// TIA Portal V17 export
// export: Created 2023-05-31T13:25:21.8623061Z, ExportSetting WithDefaults, DisplayName Totally Integrated Automation Portal, DisplayVersion V17, DisplayName TIA Portal Openness, DisplayVersion V17, DisplayName TIA Portal Version Control Interface, DisplayVersion V17, DisplayName STEP 7 Professional, DisplayVersion V17, DisplayName STEP 7 Safety, DisplayVersion V17, DisplayName WinCC Advanced, DisplayVersion V17
ORGANIZATION_BLOCK "Main"   // OB1, LAD, ProgramCycle
TITLE = "Main Program Sweep (Cycle)"
{ S7_Optimized_Access := 'TRUE' }
VERSION : 0.1
// stored: AutoNumber true, IsIECCheckEnabled false, SetENOAutomatically false
   VAR_INPUT
      Initial_Call : Bool;   // Initial call of this OB
      Remanence : Bool;   // =True, if remanent data are available
   END_VAR
BEGIN

REGION Network 1
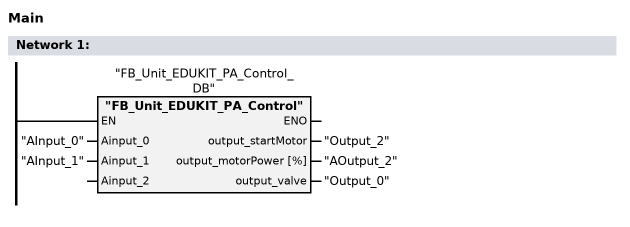
   RUNG wire#powerrail
      "FB_Unit_EDUKIT_PA_Control_DB"(Ainput_0 := "AInput_0", Ainput_1 := "AInput_1", Ainput_2 :=, output_startMotor => "Output_2", "output_motorPower [%]" => "AOutput_2", output_valve => "Output_0")
   END_RUNG
   // the same network as SCL:
   "FB_Unit_EDUKIT_PA_Control_DB"(Ainput_0 := "AInput_0",   // "FB_Unit_EDUKIT_PA_Control"
                           Ainput_1 := "AInput_1",
                           output_startMotor => "Output_2",
                           "output_motorPower [%]" => "AOutput_2",
                           output_valve => "Output_0");
END_REGION
END_ORGANIZATION_BLOCK
